// SIMATIC S7-200 project (STEP 7-Micro/WIN), CPU 224XP REL 02.01

SYMBOL_TABLE USER2
RED_1            Q0.0
YEL_1            Q0.1
GRE_1            Q0.2
RED_2            Q0.5
YEL_2            Q0.6
GRE_2            Q0.7
Delay_1          VW10
Delay_2          VW12
END_SYMBOL_TABLE

SYMBOL_TABLE S7-200 Symbols
Always_On        SM0.0    // Always ON
First_Scan_On    SM0.1    // ON for the first scan cycle only
Pot0_Value       SMB28    // Set to value corresponding to analog adjustment 0.
Pot1_Value       SMB29    // Set to value corresponding to analog adjustment 1.
END_SYMBOL_TABLE

ORGANIZATION_BLOCK MAIN:OB1
TITLE=PROGRAM COMMENTS
BEGIN
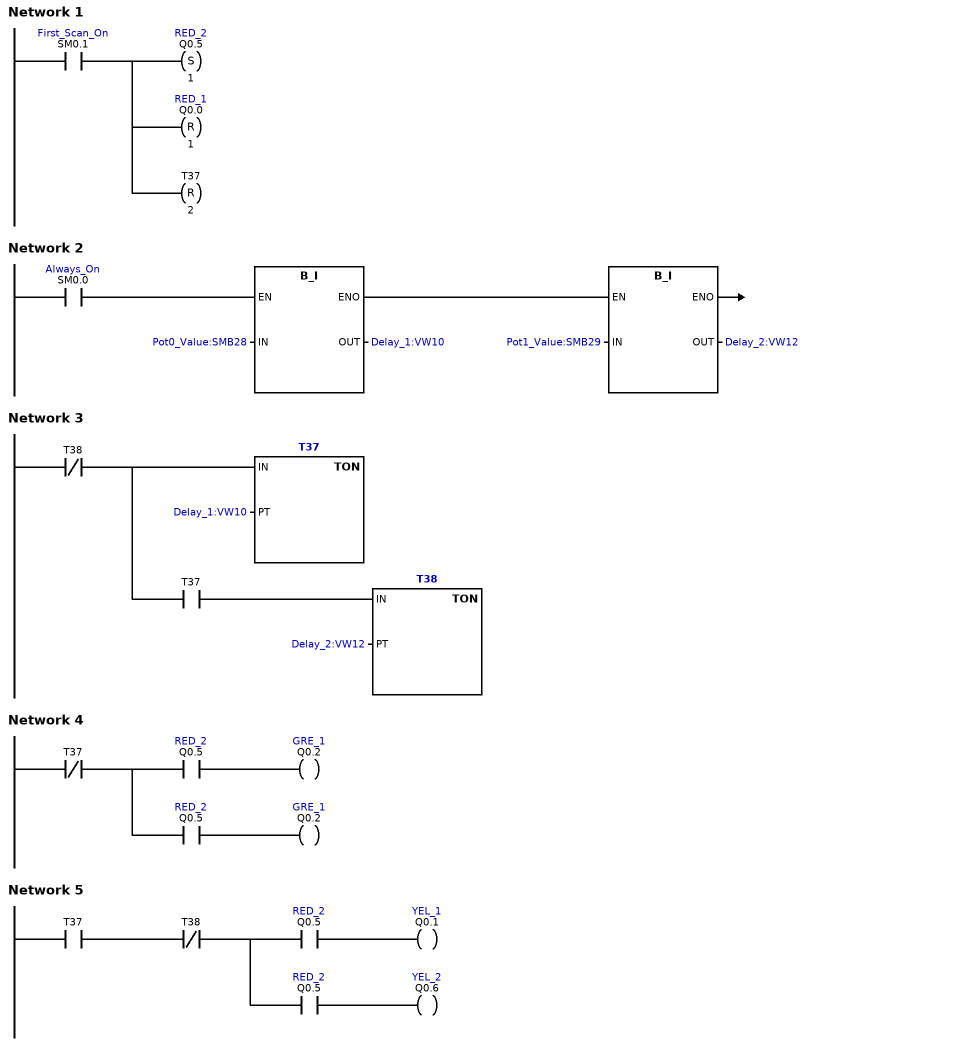
Network 1
// (network saved uncompiled; LAD cells follow)
// row 0: c0 -| |- First_Scan_On:SM0.1 v  c1 -(S) RED_2:Q0.5, 1
// row 1: c0 ^v  c1 -(R) RED_1:Q0.0, 1
// row 2: c0 ^  c1 -(R) T37, 2
Network 2
LD     Always_On:SM0.0
BTI    Pot0_Value:SMB28, Delay_1:VW10
AENO
BTI    Pot1_Value:SMB29, Delay_2:VW12
Network 3
LDN    T38
TON    T37, Delay_1:VW10
A      T37
TON    T38, Delay_2:VW12
Network 4
LDN    T37
LPS
A      RED_2:Q0.5
=      GRE_1:Q0.2
LPP
A      RED_2:Q0.5
=      GRE_1:Q0.2
Network 5
// (network saved uncompiled; LAD cells follow)
// row 0: c0 -| |- T37  c1 -|/|- T38 v  c2 -| |- RED_2:Q0.5  c3 -( ) YEL_1:Q0.1
// row 1: c1 ^  c2 -| |- RED_2:Q0.5  c3 -( ) YEL_2:Q0.6
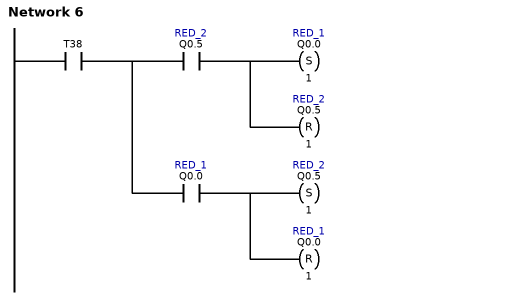
Network 6
LD     T38
LPS
A      RED_2:Q0.5
S      RED_1:Q0.0, 1
R      RED_2:Q0.5, 1
LPP
A      RED_1:Q0.0
S      RED_2:Q0.5, 1
R      RED_1:Q0.0, 1
END_ORGANIZATION_BLOCK
